FUNCTION_BLOCK FB_PV_Power_Ext_Input
VAR_INPUT PERSISTENT
	bEnable									: BOOL;													//Enable the Fuctionblock and his logic
END_VAR
VAR_INPUT
	bExtErrorPv								: BOOL;													//External Error for the Pv Function
	lrExtPvPower							: LREAL;												//External Pv power from a other Function or calculation in kW
	lrExtTotalCounterEnergy_Consumption		: LREAL;												//External Counter Value for Energy consumption with unit kWh
	lrExtTotalCounterEnergy_Production		: LREAL;												//External Counter Value for Energy production with unit kWh
	lrExtCounterEnergyT1_Consumption		: LREAL;												//External Counter Value for Energy consumption Tariff 1 with unit kWh
	lrExtCounterEnergyT2_Consumption		: LREAL;												//External Counter Value for Energy consumption Tariff 2 with unit kWh
	lrExtCounterEnergyT1_Production			: LREAL;												//External Counter Value for Energy production Tariff 1 with unit kWh
	lrExtCounterEnergyT2_Production			: LREAL;												//External Counter Value for Energy production Tariff 2 with unit kWh
END_VAR
VAR_OUTPUT
	stDataPv								: ST_PV_Output;											//{#lynus.ag#()} //Output Data Pv System
	diNrOfPv_OUT							: DINT;													//Active Number from the Pv system for using on other functions
END_VAR
VAR
	{attribute 'hide'}
	fbPv									: FB_PV_Production;										//Function block for Pv system
	{attribute 'hide'}
	fbNumberDevice							: FB_NumberOfDevice;									//Function block to calcualte the number of the Device
	fbDIErrorPv								: FB_XL1XXX_DI;											//Digital Input Error Pv System
	{attribute 'hide'}
	timDissableFunctions					: TON;													//Timer to dissable the Function after Lynus_Standards.Constants_General.tTimeDissableLynusFunctions Days without connection to the Lynus Cloud
	{attribute 'hide'}
	timResetConnectionOnGVL					: TON;													//Timer to try reset the connection Flag on the GVL. (When somebody delete the Connection Function and make only a onlinechange)
	{attribute 'hide'}
	fbPD									: FB_PersistentData_Number;								//Function to save persistent data 
	{attribute 'hide'}
	byWaitInStep							: BYTE;													//Wait in Step before start to clean data on PLC
	{attribute 'hide'}
	iStateGVLData							: INT;													//State machine to handle the data on the GVL
	{attribute 'hide'}
	diCounterForGVL							: DINT;													//Counter to clean old data on GVL
END_VAR

//Creator : Kai Ebensperger
//Company : Lynus AG
//Date : 08.06.2021
//Version : 1.0.0.0

//With this function block its possible to show the power data from a PV system.
//The Power and Error Data came from a other Function and can connect to the Inputs. The Function write the Data then on the Lynus GVL

//NOTE for diNr.....Designation => 
//_IN = Here Data come in from other Functions or go out to other functions about the GVL
//_OUT = Here Data go out to other functions about the GVL

(*-------------------------------------------------------------Calcualte the number of Pv System---------------------------------------------------------------*)

fbNumberDevice(
	diActualNumberOfDevices:= Lynus_Standards.GVL_Energy.stNumberOfDevices.diNumberOfPvSystems, 
	diMaxNumberOfDevices:= Constants_Energy.diMaxNumberOfPvSystems, 
	udiCounterOnlineChange:= TwinCAT_SystemInfoVarList._AppInfo.OnlineChangeCnt, 
	bNumberIsCalculatet=> , 
	bFPNumberIsCalculatet=> , 
	bOnlineChange=> , 
	diNumberForThisDevice=> diNrOfPv_OUT, 
	diNumberOfTotalDevices=> );

//Write new Numer on GVL
IF fbNumberDevice.bFPNumberIsCalculatet THEN
	Lynus_Standards.GVL_Energy.stNumberOfDevices.diNumberOfPvSystems := fbNumberDevice.diNumberOfTotalDevices;	
END_IF 

//Delete old Number on GVL
IF fbNumberDevice.bOnlineChange THEN 
	Lynus_Standards.GVL_Energy.stNumberOfDevices.diNumberOfPvSystems := diNrOfPv_OUT;	
		iStateGVLData := 1; 
END_IF	

(*-------------------------------------------------------------Service from Backend is ready and check the connection to backen for dissabel/enable Function---------------------------------------------------------------*)

//Try to reset the variable for connection on the GVL. When all is normal then the Lynus Mqtt connection function set this variable to true in the next cycle
//When we have no connection to the backend then after Lynus_Standards.Constants_General.tTimeDissableLynusFunctions days the Function is dissabled with all of his functionalities
timResetConnectionOnGVL(IN:= NOT timResetConnectionOnGVL.Q, PT:= T#1H, Q=> , ET=> );
	IF timResetConnectionOnGVL.Q THEN Lynus_Standards.GVL_Communicator.bStateConnectionToEnableFunctions := FALSE; END_IF
		IF NOT Lynus_Standards.GVL_Communicator.bStateConnectionToEnableFunctions THEN timDissableFunctions.IN := TRUE; ELSE timDissableFunctions.IN := FALSE; END_IF  
			timDissableFunctions(IN:= , PT:= Lynus_Standards.Constants_General.tTimeDissableLynusFunctions, Q=> , ET=> );

(*-----------------------------------------------------------------------------Error ----------------------------------------------------------------------------*)

fbDIErrorPv(bInvers:= FALSE, bSignal=> );	

IF timDissableFunctions.Q THEN fbPv.bWarning := TRUE; fbPv.iWarningCode := 0; ELSE fbPv.bWarning := FALSE; END_IF 	
	IF fbDIErrorPv.bSignal OR Lynus_Standards.GVL_Energy.stNumberOfDevices.diNumberOfPvSystems > Constants_Energy.diMaxNumberOfPvSystems OR bExtErrorPv THEN fbPv.bError := TRUE; ELSE fbPv.bError := FALSE; END_IF 
		//Error Code
		IF Lynus_Standards.GVL_Energy.stNumberOfDevices.diNumberOfPvSystems > Constants_Energy.diMaxNumberOfPvSystems THEN fbPv.iErrorCode := 1; END_IF  
		IF fbDIErrorPv.bSignal OR bExtErrorPv THEN fbPv.iErrorCode := 0; END_IF 

fbPv(
	bEnable:= bEnable AND NOT timDissableFunctions.Q, 
	bError:= , 
	bWriteWithDelay:= TRUE, 
	iErrorCode:= , 
	iWarningCode:= , 
	lrTotalCounterEnergy_Consumption:= lrExtTotalCounterEnergy_Consumption * 1000, 
	lrTotalCounterEnergy_Production:= lrExtTotalCounterEnergy_Production * 1000, 
	lrCounterEnergyT1_Consumption:= lrExtCounterEnergyT1_Consumption * 1000, 
	lrCounterEnergyT2_Consumption:= lrExtCounterEnergyT2_Consumption * 1000, 
	lrCounterEnergyT1_Production:= lrExtCounterEnergyT1_Production * 1000, 
	lrCounterEnergyT2_Production:= lrExtCounterEnergyT2_Production * 1000, 
	lrPvPower:= lrExtPvPower * 1000, 
	tTimDelayOutput:= T#5S, 
	stDataPvOut=> , 
	stDataPvOutDelay=> stDataPv);	
		
(*-----------------------------------------------------------Handle data to Global structure for the Pv system-----------------------------------------------------------------*)

CASE iStateGVLData OF
	
	0://Init Step
		byWaitInStep := 0;
			diCounterForGVL := 1;
	
	1://Wait for 4 Steps before clean al Data on GVL
		byWaitInStep := byWaitInStep + 1;
			IF byWaitInStep >= 4 AND fbNumberDevice.bNumberIsCalculatet THEN iStateGVLData := 2; END_IF
				//To much Devices, back to the Init step
				IF byWaitInStep >= 4 AND NOT fbNumberDevice.bNumberIsCalculatet THEN iStateGVLData := 0; END_IF	
			
	2://Clear all Data in GVL
		Lynus_Standards.GVL_Energy.stDataOfPvSystems[diCounterForGVL].bEnabled := FALSE;
			Lynus_Standards.GVL_Energy.stDataOfPvSystems[diCounterForGVL].byErrorWarning := 0;
				Lynus_Standards.GVL_Energy.stDataOfPvSystems[diCounterForGVL].lrPowerConsumption := 0;
					Lynus_Standards.GVL_Energy.stDataOfPvSystems[diCounterForGVL].lrPower := 0;
						Lynus_Standards.GVL_Energy.stDataOfPvSystems[diCounterForGVL].lrPowerProduction := 0;	
		
		diCounterForGVL := diCounterForGVL + 1;
			diCounterForGVL := LIMIT(0,diCounterForGVL,Constants_Energy.diMaxNumberOfPvSystems);
				//Back to the init step
				IF diCounterForGVL >= Constants_Energy.diMaxNumberOfPvSystems THEN iStateGVLData := 0; END_IF

END_CASE 	 

IF diNrOfPv_OUT > 0 AND fbNumberDevice.bNumberIsCalculatet THEN
	Lynus_Standards.GVL_Energy.stDataOfPvSystems[diNrOfPv_OUT].bEnabled := fbPv.stDataPvOut.bEnabled;
		Lynus_Standards.GVL_Energy.stDataOfPvSystems[diNrOfPv_OUT].byErrorWarning := fbPv.stDataPvOut.byErrorWarning;
			Lynus_Standards.GVL_Energy.stDataOfPvSystems[diNrOfPv_OUT].lrPowerConsumption := fbPv.stDataPvOut.lrPowerConsumption;
				Lynus_Standards.GVL_Energy.stDataOfPvSystems[diNrOfPv_OUT].lrPower := fbPv.stDataPvOut.lrPower;
					Lynus_Standards.GVL_Energy.stDataOfPvSystems[diNrOfPv_OUT].lrPowerProduction := fbPv.stDataPvOut.lrPowerProduction;
END_IF

(*----------------------------------------------------------Save persistent data----------------------------------------------------------------*)

fbPD(lrValue:= BOOL_TO_LREAL(bEnable), bEventBasedActive=> );

END_FUNCTION_BLOCK

(* stored: Version 1.1.0.1, ProductVersion 3.1.4024.9
   POU FB_PV_Power_Ext_Input: Id {07b02d87-5281-476f-b119-657fdaec310e}, SpecialFunc None *)
